// TIA Portal V16 export
// export: Created 2020-03-17T19:17:40.9648314Z, ExportSetting None, DisplayName Totally Integrated Automation Portal, DisplayVersion V16, DisplayName TIA Portal Version Control Interface, DisplayVersion V16, DisplayName TIA Portal Openness, DisplayVersion V16, DisplayName STEP 7 Professional, DisplayVersion V16, DisplayName STEP 7 Safety, DisplayVersion V16, DisplayName WinCC Advanced, DisplayVersion V16
FUNCTION "Baustein_1" : Void   // FC1, LAD
{ S7_Optimized_Access := 'TRUE' }
// stored: SetENOAutomatically false
BEGIN
END_FUNCTION
